FUNCTION_BLOCK UNIT_StateManager (* Unit state manager: OPC UA methods Reset/Start/Clear(Session) answer [Accepted, ErrorID]; publishes the PackML State; EXECUTE starts the Execute procedure *)
  (* Standard: 61499-2 *)
  (* Version 0.1, 2026-09-28, Project contributors, AAU Smart Production Lab *)
  PACKAGE unitlib;
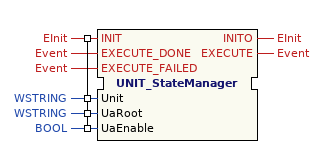
  EVENT_INPUT
    INIT : EInit WITH Unit, UaRoot, UaEnable;
    EXECUTE_DONE;
    EXECUTE_FAILED;
  END_EVENT
  EVENT_OUTPUT
    INITO : EInit;
    EXECUTE;
  END_EVENT
  VAR_INPUT
    Unit : WSTRING;
    UaRoot : WSTRING;
    UaEnable : BOOL;
  END_VAR
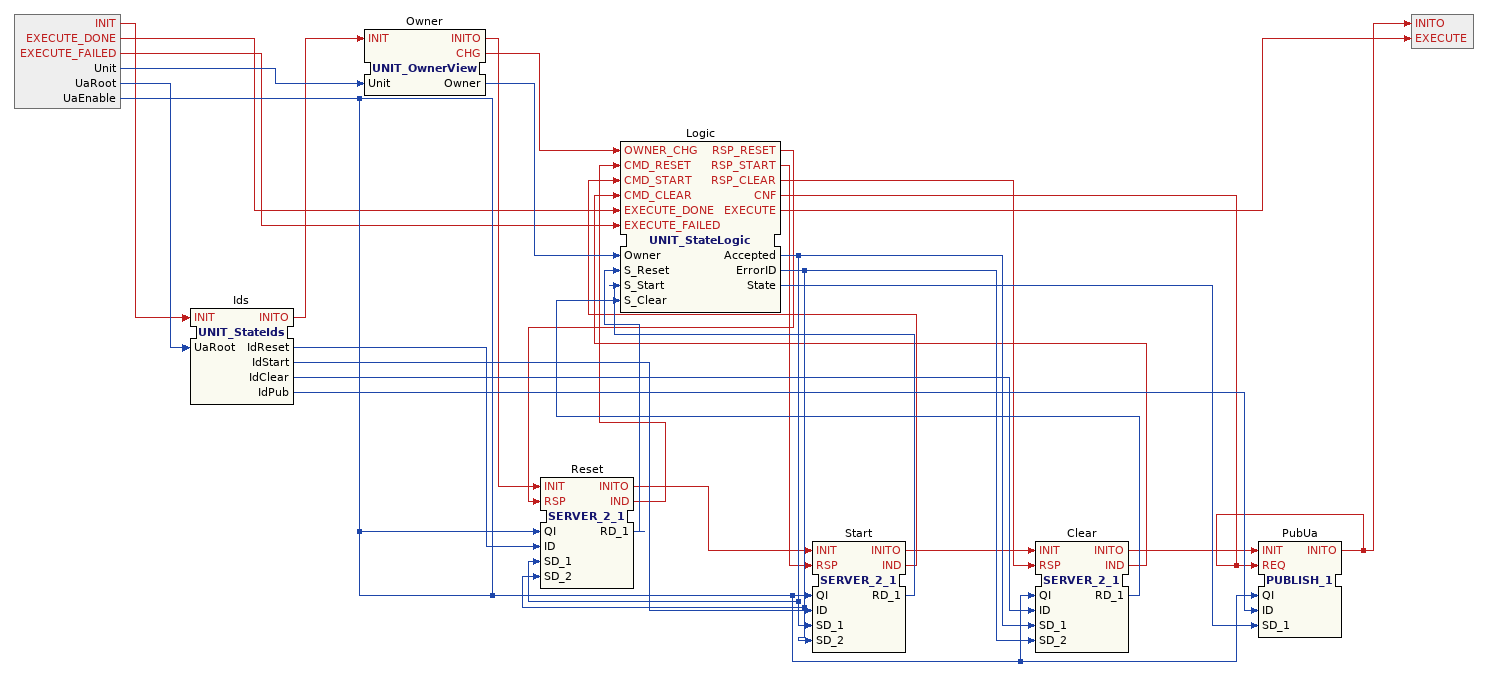
  FBS
    Ids : unitlib::UNIT_StateIds;
    Owner : unitlib::UNIT_OwnerView;
    Reset : iec61499::net::SERVER_2_1;
    Start : iec61499::net::SERVER_2_1;
    Clear : iec61499::net::SERVER_2_1;
    Logic : unitlib::UNIT_StateLogic;
    PubUa : iec61499::net::PUBLISH_1;
  END_FBS
  EVENT_CONNECTIONS
    INIT TO Ids.INIT;
    Ids.INITO TO Owner.INIT;
    Owner.INITO TO Reset.INIT;
    Reset.INITO TO Start.INIT;
    Start.INITO TO Clear.INIT;
    Clear.INITO TO PubUa.INIT;
    PubUa.INITO TO PubUa.REQ;
    PubUa.INITO TO INITO;
    Owner.CHG TO Logic.OWNER_CHG;
    Reset.IND TO Logic.CMD_RESET;
    Logic.RSP_RESET TO Reset.RSP;
    Start.IND TO Logic.CMD_START;
    Logic.RSP_START TO Start.RSP;
    Clear.IND TO Logic.CMD_CLEAR;
    Logic.RSP_CLEAR TO Clear.RSP;
    Logic.CNF TO PubUa.REQ;
    Logic.EXECUTE TO EXECUTE;
    EXECUTE_DONE TO Logic.EXECUTE_DONE;
    EXECUTE_FAILED TO Logic.EXECUTE_FAILED;
  END_CONNECTIONS
  DATA_CONNECTIONS
    UaRoot TO Ids.UaRoot;
    Unit TO Owner.Unit;
    UaEnable TO Reset.QI;
    UaEnable TO Start.QI;
    UaEnable TO Clear.QI;
    UaEnable TO PubUa.QI;
    Owner.Owner TO Logic.Owner;
    Ids.IdReset TO Reset.ID;
    Reset.RD_1 TO Logic.S_Reset;
    Logic.Accepted TO Reset.SD_1;
    Logic.ErrorID TO Reset.SD_2;
    Ids.IdStart TO Start.ID;
    Start.RD_1 TO Logic.S_Start;
    Logic.Accepted TO Start.SD_1;
    Logic.ErrorID TO Start.SD_2;
    Ids.IdClear TO Clear.ID;
    Clear.RD_1 TO Logic.S_Clear;
    Logic.Accepted TO Clear.SD_1;
    Logic.ErrorID TO Clear.SD_2;
    Ids.IdPub TO PubUa.ID;
    Logic.State TO PubUa.SD_1;
  END_CONNECTIONS
END_FUNCTION_BLOCK
